(* CODESYS project EAS SCADA.library
   Author: EAS
   Placeholder: EAS SCADA
   Title: EAS SCADA
   Version: 1.0.4
   Company: ESCARRE AUTOMATIZACION Y SERVICIOS sl

Project tree, tasks and I/O mapping:
  libraries: Tc2_Standard, * (Beckhoff Automation GmbH); Tc2_System, * (Beckhoff Automation GmbH); Tc3_Module, * (Beckhoff Automation GmbH)
  DUTs/
    PE/
      data type E_Funcio
      data type PasCicle
      data type T_Compat
      data type T_funcio
      data type T_Sirena
  GVLs/
    global variables Batch
    global variables CONSTANTS
  POUs/
    BATCH/
      function block CarregarFuncionsActivesAlDB [ST]
      function block ComprobarFuncionsPas [ST]
      function block Inic_Func_Actv [ST]
      function block Parar_Func_FiFuncio [ST]
      function block Parar_Func_Incomp [ST]
      function block PararTotesLesFuncions [ST]
      function block Salt [ST]
      function block SaltDePasEnUnCicle [ST]
    GestioPE/
      function block Alarma_v01 [ST]
      function block FunBck_v01 [ST]
      function block Func_Activa_v01 [ST]
  VISUs/
*)

// DUTs/PE/E_Funcio
TYPE E_Funcio :
STRUCT

	Cd_Funcio:WORD;
	Actv_Funcio:BOOL;
	ParamFunc:ARRAY [1..Max_ParamFunc] OF WORD;

END_STRUCT
END_TYPE

// DUTs/PE/PasCicle
TYPE PasCicle :
STRUCT
	Pas:WORD;
	Funcio:E_Funcio;

END_STRUCT
END_TYPE

// DUTs/PE/T_Compat
TYPE T_Compat :
STRUCT

	Funcio1:WORD;  			(*Codi de la primera funcio*)
	Funcio2:WORD;  			(*Codi de la segona funcio*)

END_STRUCT
END_TYPE

// DUTs/PE/T_funcio
TYPE T_funcio :
STRUCT

	Cd_funcio:WORD;												(*Codi de la funció*)
	DesFuncio:STRING(16);										(*Descripció de la funció*)
	Background:BOOL;												(*Indicació per si la funció es en backgraund o no*)
	FinFunc:ARRAY [1..max_FinFunc] OF WORD;					(*Funcions que s'han d'acabar al començar aquesta*)

END_STRUCT
END_TYPE

// DUTs/PE/T_Sirena
TYPE T_Sirena :
STRUCT
	Actv:BOOL;
	Rearme:BOOL;
END_STRUCT
END_TYPE

// GVLs/Batch

VAR_GLOBAL RETAIN

(*=======================================	*)
(*					Estat del PE4							*)
(*=======================================	*)

(*Estat de PE4*)
	Func_Comp: ARRAY [1..Max_Compatibles] OF T_Compat;


(*=======================================	*)
(*			Variables de gestió de funcions				*)
(*=======================================	*)

(*Estat de lesFuncions *)
	Est_Func: ARRAY [1..Max_Funcions] OF E_Funcio;  		(*Estat actual de les funcions*)
	Est_F_PE4: ARRAY [1..Max_Funcions] OF E_Funcio;  		(*Estat de les funcions per les comunicacions del PE4*)
	Est_F_PE4_Ant: ARRAY [1..Max_Funcions] OF E_Funcio;  	(*Estat de les funcions per les comunicacions del PE4*)


(* *)
	Config_Func: ARRAY  [1..Max_Funcions] OF t_funcio;		(*Configuració de les funcios *)
	Config_Func_Ampl: ARRAY  [1..Max_Funcions] OF t_funcio_Ampl;		(*Configuració de les funcios ampliades*)
	Func_Actives: ARRAY [1..Max_Func_Pas] OF WORD;		(* DB que indica en automaatic les funcions que estan en marcha en automatic*)


(*=======================================	*)
(*			Variables de gestió de cicle					*)
(*=======================================	*)

(*Cicles*)
	Cicle0: ARRAY [1..max_PasCicle] OF PasCicle;  			(*Cicle Actual de treball*)
	CicleRebut: ARRAY [1..max_PasCicle] OF PasCicle;  		(*Cicle Rebut*)


(*=======================================	*)
(*					Alarmes								*)
(*=======================================	*)

	Alarmes:ARRAY[1..Max_Alarmes] OF T_Alarma;
	Sirena:ARRAY[1..Max_Alarmes] OF T_Sirena;


(*=======================================	*)
(*			Parametres fixes								*)
(*=======================================	*)

	ParamFixes:ARRAY[1..Max_ParamFixes] OF T_ParamFixe;


(*=======================================	*)
(*			Botons Auto/Man								*)
(*=======================================	*)

	PulsadorManual:BOOL;
	PulsadorAutomatic:BOOL;

(*=======================================	*)
(*			Marcas Internes								*)
(*=======================================	*)

	InicioCiclo:BOOL;


END_VAR


VAR_GLOBAL

(*=======================================	*)
(*			Maquina paralel 								*)
(*=======================================	*)

	TipoParalelo:WORD;
	MaquinaEnParalel:BOOL:=FALSE;
	Master:BOOL;
	Slave:BOOL;
	Pas_M:DWORD;
	Pas_S1:DWORD;
	Pas_S2:DWORD;
	Pas_S3:DWORD;
	Pas_S4:DWORD;
	Tipus_P:DWORD;
	Preparat_C_local:BOOL;
	He_C_local:BOOL;
	Ordre_C:BOOL;
	Ordre_C_Master:BOOL;
	Preparat_C_S1:BOOL;
	Preparat_C_S2:BOOL;
	Preparat_C_S3:BOOL;
	Preparat_C_S4:BOOL;
	He_C_S1:BOOL;
	He_C_S2:BOOL;
	He_C_S3:BOOL;
	He_C_S4:BOOL;
	Fi_C:BOOL;
	Fi_C_master:BOOL;



(*			CONSERVAR  COMPATIBILITAT				*)

	EsperaParalelPerSaltar:BOOL;
	SaltdePas:BOOL;


END_VAR

// GVLs/CONSTANTS

VAR_GLOBAL CONSTANT

(*=======================================	*)
(*			Carregar Constants						*)
(*=======================================	*)
	Max_Funcions:WORD:=64;
	Max_ParamFunc:WORD:=9;
	max_FinFunc:WORD:=5;
	max_PasCicle:WORD:=256;
	Max_Compatibles:WORD:=32;
	Max_Func_Pas:WORD:=12;
	Max_Alarmes:WORD:=128;
	Max_ParamFixes:WORD:=150;
	Max_DBFiFuncio: WORD:=320 ;				(* Es calcula com    (Max_Funcions*Max_FinFunc)   *)
	Max_ElementsCicle: WORD:=2816 ;		(* Es calcula com    (Max_PasCicle*(Max_ParamFunc+2))  *)
	Max_DBIncompatibles: WORD:=64;			(* Es calcula com    (Max_Compatibles*2)  *)
	Max_Inputs: WORD:=128;
	Max_Outputs: WORD:=128;
	Max_Analog: WORD:=32;
	Num_Prod_Dos:WORD:=10;         					(* Numero maximo de productos en una dosificación*)
	Max_Prod_Dos:WORD:=128;							(* Productos en una dosificadora*)
	Max_Valv_Dos:WORD:=128;							(* Valvulas en una dosificadora*)
END_VAR

// POUs/BATCH/CarregarFuncionsActivesAlDB
FUNCTION_BLOCK CarregarFuncionsActivesAlDB

(***********************************************************************
Aquest Bloc Carrega les Funcions actives al "DB d'estat de les funcions"
al "DB de funcions actives".   
************************************************************************)

VAR_INPUT
	EstatFuncions: ARRAY [1..max_funcions] OF E_Funcio;
END_VAR

VAR_OUTPUT
	FuncionsActives:ARRAY [1..Max_Func_Pas] OF WORD;
END_VAR

VAR
	Punter:WORD;
	PunterDB:WORD;
	inicialitzaDB: Inic_Func_Actv;
	DB_ple: BOOL;

END_VAR

inicialitzaDB(Func_Actv:= FuncionsActives);
DB_Ple:=FALSE;
punter:=1;
punterDB:=1;
WHILE (punter<=max_funcions)AND NOT(DB_Ple)
	DO
		IF EstatFuncions[punter].Actv_Funcio
			THEN
				FuncionsActives[PunterDB]:=EstatFuncions[punter].Cd_Funcio;
				PunterDB:=PunterDB+1;
				IF punterDB>Max_Func_Pas
					THEN
						DB_ple:=TRUE;
				END_IF
		END_IF
		punter:=punter+1;
END_WHILE

END_FUNCTION_BLOCK

// POUs/BATCH/Inic_Func_Actv
FUNCTION_BLOCK Inic_Func_Actv

(*********************************************************
Reinicia el DB de les funcions actives
***********************************************************)

VAR_IN_OUT
	Func_Actv: ARRAY [1..Max_Func_Pas] OF WORD;		(* DB que indica en automaatic les funcions que estan en marcha en automatic*)
END_VAR

VAR
	Punter: WORD;
END_VAR

Punter:=1;

REPEAT
	Func_Actv[punter]:=0;
	Punter:=Punter+1;
UNTIL
	Punter>Max_Func_Pas
END_REPEAT

END_FUNCTION_BLOCK

// POUs/BATCH/ComprobarFuncionsPas
FUNCTION_BLOCK ComprobarFuncionsPas

(************************************************************
Aquest Bloc Comproba les funcions actves que hi ha en aquest
pas i quan acaben dona l'ordr de canviar de pas.
**************************************************************)

VAR_INPUT
	Estat_F: ARRAY [1..Max_Funcions] OF E_Funcio;
	Tipus_F:ARRAY [1..Max_Funcions] OF T_Funcio;
	FuncionsActives:ARRAY [1..Max_Func_Pas] OF WORD;
END_VAR

VAR_OUTPUT
	AumentaPas:BOOL;
END_VAR

VAR
	Punter: WORD;
	Aumenta: BOOL;
	TempoPAS:TON;

END_VAR

(*Inicialitzar els punters*)
Punter:=1;
Aumenta:=TRUE;

REPEAT
	IF (FuncionsActives[Punter]<>0)AND((Estat_F[FuncionsActives[Punter]].Actv_Funcio=TRUE)AND(Tipus_F[FuncionsActives[Punter]].Background=FALSE))
		THEN
			Aumenta:=FALSE;
	END_IF
	Punter:=Punter+1;
UNTIL
	(Punter>Max_Func_Pas)OR(Aumenta=FALSE)
END_REPEAT

TempoPAS
	(IN:=Aumenta ,
	PT:=t#500ms ,
	Q=>AumentaPas ,
	ET=> );

END_FUNCTION_BLOCK

// POUs/BATCH/Parar_Func_FiFuncio
FUNCTION_BLOCK Parar_Func_FiFuncio

(**************************************************
Para les funcions del "DB de l'estat de funcions" 
depenen de la funcio de la entreda per "fifuncion"
***************************************************)

VAR_INPUT
	Tipus_Funcio:T_funcio;
END_VAR
VAR_OUTPUT
END_VAR
VAR_IN_OUT
	Estat_F: ARRAY [1..Max_Funcions] OF E_Funcio;
END_VAR
VAR
	PunterFiFunc:WORD;
	FuncioIncompat: WORD;
END_VAR

(*..................	Parar les funcions per fin función..................................	*)
PunterFiFunc:=1;
WHILE (PunterFiFunc <= max_FinFunc) DO
	FuncioIncompat :=Tipus_funcio.FinFunc[PunterFiFunc];
	IF FuncioIncompat <>0
		THEN
			Estat_F [FuncioIncompat].Actv_Funcio:=FALSE;
	END_IF
	PunterFiFunc:=PunterFiFunc+1;
END_WHILE

END_FUNCTION_BLOCK

// POUs/BATCH/Parar_Func_Incomp
FUNCTION_BLOCK Parar_Func_Incomp
(************************************************************
L'hi introduim una funció i el el bloc para les funcions del 
"DB estat de les funcions" depenen del 
"DB de compatibilitat"
**************************************************************)
VAR_INPUT
	Funcio:WORD;  (*Funcio que s'ha de parar*)
END_VAR

VAR_OUTPUT
END_VAR

VAR_IN_OUT
	DB_Comp:ARRAY [1..Max_Compatibles] OF T_Compat;
	Estat_F: ARRAY [1..Max_Funcions] OF E_Funcio;
END_VAR

VAR
	PunterEstat:WORD;
	PunterComp:WORD;
END_VAR

(*Mirar si hi ha alguna funció incompatible amb la nova funció*)
PunterEstat:=1;
PunterComp:=1;
REPEAT
	IF DB_Comp[PunterComp].Funcio1=Funcio
		THEN
			PunterEstat:=DB_Comp[PunterComp].Funcio2;
			Estat_F[PunterEstat].Actv_Funcio:=FALSE;
	END_IF
	PunterComp:=PunterComp+1;
UNTIL
	(PunterComp>Max_Compatibles)
END_REPEAT

END_FUNCTION_BLOCK

// POUs/BATCH/PararTotesLesFuncions
FUNCTION_BLOCK PararTotesLesFuncions
(********************************************************
Parar totes les funcions del "DB estat"
*********************************************************)
VAR_IN_OUT
	Estat_F: ARRAY [1..Max_Funcions] OF E_Funcio;
END_VAR

VAR
	Punter: WORD;
END_VAR

(*Inicialitzar els punters*)
Punter:=1;


WHILE (Punter <= Max_Funcions) DO
	IF Estat_F[Punter].Actv_Funcio=TRUE
		THEN
			Estat_F [Punter].Actv_Funcio:=FALSE;
	END_IF
	Punter:=Punter+1;
END_WHILE

END_FUNCTION_BLOCK

// POUs/BATCH/Salt
FUNCTION_BLOCK Salt
(************************************************************
Salta del "Pas inicial" al "Pas Final"  del  "BDCicle"
**************************************************************)
VAR_INPUT
	PasInicial:DWORD;
	PasFinal:DWORD;
END_VAR

VAR_IN_OUT


END_VAR

VAR

	FIFuncio:Parar_Func_FiFuncio;
	Incompatibles:Parar_Func_Incomp;
	PunterCicle:WORD;					(* Aquest valor marca la popsició del db de cicle on estem independent del pas de cicle *)
	T_Func_Act:T_Funcio;				(* Funcio que indica el punterCicle *)

	codi: WORD;

	Est_Func_0: ARRAY [1..Max_Funcions] OF E_Funcio;  		(*Estat de les funcions a cero per reiniciar l'estat*)
END_VAR

(*,,,,,,,,,,,,,,,,,,,,Carregar la posició inicial depenen si es salta desde:
				el pas cero: carerega d'un cicle nou
				un pas en concret: salt sobre el cicle que ja està carregat ,,,,,,,,,,,,,,,,,,,,,  *)

IF PasInicial=0
	THEN
		(*Posar Punter al primer pas*)
		PunterCicle:=1;
		(*Inicialitzar el estat de les funcions*)
		Est_Func:=Est_Func_0;
	ELSE
		(*Buscar Punter Cicle del pas inicial*)
		PunterCicle:=0;
		REPEAT
			PunterCicle := PunterCicle+1;
		UNTIL
			(((Cicle0[PunterCicle].Pas=PasInicial)AND(Cicle0[PunterCicle+1].Pas<>PasInicial)) OR (PunterCicle>=max_PasCicle))
		END_REPEAT
		PunterCicle := PunterCicle+1;      (*02/06/05*)
END_IF

(*,,,,,,,,,,,,,,,,,,,,Bucle de control,,,,,,,,,,,,,,,,,,,,,,,,,,,,,,,,,,,,,,,,,,,,,,,,,,,,,,,,,,,,,	*)

REPEAT
(*.................. Carregar la funció del pas............................................. *)
		codi:=Cicle0[PunterCicle].Funcio.Cd_Funcio;
		IF codi<>0 THEN
		T_Func_Act:=Config_Func[codi];
		END_IF
(*..................	Parar les funcions incompatibles..................................	*)
		Incompatibles(
			Funcio:=T_Func_Act.Cd_funcio ,
			DB_Comp:= Func_Comp ,
			Estat_F:= Est_Func );

(*..................	Activar si es en Background ........................................	*)
		IF T_Func_Act.Background=TRUE
			THEN
				Est_Func[T_Func_Act.Cd_Funcio] := Cicle0[PunterCicle].Funcio ; 	(*Carregar parametres*)
				Est_Func[T_Func_Act.Cd_Funcio].Actv_Funcio:=TRUE;			(*Posar la funció en actiu*)
		END_IF

(*..................	Parar les funcions per fin función..................................	*)
		FiFuncio(
			Tipus_Funcio:=  T_Func_Act ,
			 Estat_F:=Est_Func	 );

(*,,,,,,,,,,,,,,,,,,	Activar funció,,,,,,,,,,,,,,,,,,,,,,,,,,,,,,,,,,,,,,,,,,,,,,,,,,,,,,,,,,,,,,,,,,,	*)
		IF Cicle0[PunterCicle].Pas = PasFinal
			THEN
				Est_Func[T_Func_Act.Cd_Funcio] := Cicle0[PunterCicle].Funcio ;	(*Carregar parametres*)
				Est_Func[T_Func_Act.Cd_Funcio].Actv_Funcio := TRUE;			(*Posar la funció en actiu*)
		END_IF

(*,,,,,,,,,,,,,,,,,,Aumentar el Punter del cicle,,,,,,,,,,,,,,,,,,,,,,,,,,,,,,,,,,,,,,,,,,	*)
		PunterCicle := PunterCicle+1;

UNTIL
	(((Cicle0[PunterCicle].Pas <> PasFinal)AND(Cicle0[PunterCicle-1].Pas = PasFinal))
	OR(PunterCicle>max_PasCicle)
	OR(Cicle0[PunterCicle-1].Funcio.Cd_Funcio=0))
END_REPEAT

END_FUNCTION_BLOCK

// POUs/BATCH/SaltDePasEnUnCicle
FUNCTION_BLOCK SaltDePasEnUnCicle
(************************************************************
Salta del "Pas inicial" al "Pas Final"  del  "BDCicle"
**************************************************************)
VAR_INPUT
	PasInicial:DWORD;
	PasFinal:DWORD;
END_VAR

VAR_IN_OUT


END_VAR

VAR

	FIFuncio:Parar_Func_FiFuncio;
	Incompatibles:Parar_Func_Incomp;
	PunterCicle:WORD;					(* Aquest valor marca la popsició del db de cicle on estem independent del pas de cicle *)
	T_Func_Act:T_Funcio;				(* Funcio que indica el punterCicle *)

	codi: WORD;

	Est_Func_0: ARRAY [1..Max_Funcions] OF E_Funcio;  		(*Estat de les funcions a cero per reiniciar l'estat*)
END_VAR

(*,,,,,,,,,,,,,,,,,,,,Carregar la posició inicial depenen si es salta desde:
				el pas cero: carerega d'un cicle nou
				un pas en concret: salt sobre el cicle que ja està carregat ,,,,,,,,,,,,,,,,,,,,,  *)

IF PasInicial=0
	THEN
		(*Posar Punter al primer pas*)
		PunterCicle:=1;
		(*Inicialitzar el estat de les funcions*)
		Est_Func:=Est_Func_0;
	ELSE
		(*Buscar Punter Cicle del pas inicial*)
		PunterCicle:=0;
		REPEAT
			PunterCicle := PunterCicle+1;
		UNTIL
			(((Cicle0[PunterCicle].Pas=PasInicial)AND(Cicle0[PunterCicle+1].Pas<>PasInicial)) OR (PunterCicle>=max_PasCicle))
		END_REPEAT
		PunterCicle := PunterCicle+1;      (*02/06/05*)
END_IF

(*,,,,,,,,,,,,,,,,,,,,Bucle de control,,,,,,,,,,,,,,,,,,,,,,,,,,,,,,,,,,,,,,,,,,,,,,,,,,,,,,,,,,,,,	*)

REPEAT
(*.................. Carregar la funció del pas............................................. *)
		codi:=Cicle0[PunterCicle].Funcio.Cd_Funcio;
		IF codi<>0 THEN
		T_Func_Act:=Config_Func[codi];
		END_IF
(*..................	Parar les funcions incompatibles..................................	*)
		Incompatibles(
			Funcio:=T_Func_Act.Cd_funcio ,
			DB_Comp:= Func_Comp ,
			Estat_F:= Est_Func );

(*..................	Activar si es en Background ........................................	*)
		IF T_Func_Act.Background=TRUE
			THEN
				Est_Func[T_Func_Act.Cd_Funcio] := Cicle0[PunterCicle].Funcio ; 	(*Carregar parametres*)
				Est_Func[T_Func_Act.Cd_Funcio].Actv_Funcio:=TRUE;			(*Posar la funció en actiu*)
		END_IF

(*..................	Parar les funcions per fin función..................................
		FiFuncio(
			Tipus_Funcio:=  T_Func_Act ,
			 Estat_F:=Est_Func	 );										*)

(*,,,,,,,,,,,,,,,,,,	Activar funció,,,,,,,,,,,,,,,,,,,,,,,,,,,,,,,,,,,,,,,,,,,,,,,,,,,,,,,,,,,,,,,,,,,	*)
		IF Cicle0[PunterCicle].Pas = PasFinal
			THEN
				Est_Func[T_Func_Act.Cd_Funcio] := Cicle0[PunterCicle].Funcio ;	(*Carregar parametres*)
				Est_Func[T_Func_Act.Cd_Funcio].Actv_Funcio := TRUE;			(*Posar la funció en actiu*)
		END_IF

(*,,,,,,,,,,,,,,,,,,Aumentar el Punter del cicle,,,,,,,,,,,,,,,,,,,,,,,,,,,,,,,,,,,,,,,,,,	*)
		PunterCicle := PunterCicle+1;

UNTIL
	(((Cicle0[PunterCicle].Pas <> PasFinal)AND(Cicle0[PunterCicle-1].Pas = PasFinal))
	OR(PunterCicle>max_PasCicle)
	OR(Cicle0[PunterCicle-1].Funcio.Cd_Funcio=0))
END_REPEAT

END_FUNCTION_BLOCK

// POUs/GestioPE/Alarma_v01
FUNCTION_BLOCK Alarma_v01

(******************************************************
Aquest Bloc serveix per reactivar les senyals d'alarma
treballa amb el DB Sirena
********************************************************)

VAR_INPUT
END_VAR
VAR_OUTPUT
	ReactivaAlarma: BOOL;
	AlarmaActv: BOOL;
END_VAR

VAR_IN_OUT
END_VAR

VAR
	PolsA1:R_TRIG;
	PolsA2:R_TRIG;
	PolsA3:R_TRIG;
	PolsA4:R_TRIG;
	PolsA5:R_TRIG;
	PolsA6:R_TRIG;
	PolsA7:R_TRIG;
	PolsA8:R_TRIG;
	PolsA9:R_TRIG;
	PolsA10:R_TRIG;
	PolsA11:R_TRIG;
	PolsA12:R_TRIG;
	PolsA13:R_TRIG;
	PolsA14:R_TRIG;
	PolsA15:R_TRIG;
	PolsA16:R_TRIG;
	PolsA17:R_TRIG;
	PolsA18:R_TRIG;
	PolsA19:R_TRIG;
	PolsA20:R_TRIG;
	PolsA21:R_TRIG;
	PolsA22:R_TRIG;
	PolsA23:R_TRIG;
	PolsA24:R_TRIG;
	PolsA25:R_TRIG;
	PolsA26:R_TRIG;
	PolsA27:R_TRIG;
	PolsA28:R_TRIG;
	PolsA29:R_TRIG;
	PolsA30:R_TRIG;
	PolsA31:R_TRIG;
	PolsA32:R_TRIG;
	PolsA33:R_TRIG;
	PolsA34:R_TRIG;
	PolsA35:R_TRIG;
	PolsA36:R_TRIG;
	PolsA37:R_TRIG;
	PolsA38:R_TRIG;
	PolsA39:R_TRIG;
	PolsA40:R_TRIG;
	PolsA41:R_TRIG;
	PolsA42:R_TRIG;
	PolsA43:R_TRIG;
	PolsA44:R_TRIG;
	PolsA45:R_TRIG;
	PolsA46:R_TRIG;
	PolsA47:R_TRIG;
	PolsA48:R_TRIG;
	PolsA49:R_TRIG;
	PolsA50:R_TRIG;
	PolsA51:R_TRIG;
	PolsA52:R_TRIG;
	PolsA53:R_TRIG;
	PolsA54:R_TRIG;
	PolsA55:R_TRIG;
	PolsA56:R_TRIG;
	PolsA57:R_TRIG;
	PolsA58:R_TRIG;
	PolsA59:R_TRIG;
	PolsA60:R_TRIG;
	PolsA61:R_TRIG;
	PolsA62:R_TRIG;
	PolsA63:R_TRIG;
	PolsA64:R_TRIG;
	PolsA65:R_TRIG;
	PolsA66:R_TRIG;
	PolsA67:R_TRIG;
	PolsA68:R_TRIG;
	PolsA69:R_TRIG;
	PolsA70:R_TRIG;
	PolsA71:R_TRIG;
	PolsA72:R_TRIG;
	PolsA73:R_TRIG;
	PolsA74:R_TRIG;
	PolsA75:R_TRIG;
	PolsA76:R_TRIG;
	PolsA77:R_TRIG;
	PolsA78:R_TRIG;
	PolsA79:R_TRIG;
	PolsA80:R_TRIG;
	PolsA81:R_TRIG;
	PolsA82:R_TRIG;
	PolsA83:R_TRIG;
	PolsA84:R_TRIG;
	PolsA85:R_TRIG;
	PolsA86:R_TRIG;
	PolsA87:R_TRIG;
	PolsA88:R_TRIG;
	PolsA89:R_TRIG;
	PolsA90:R_TRIG;
	PolsA91:R_TRIG;
	PolsA92:R_TRIG;
	PolsA93:R_TRIG;
	PolsA94:R_TRIG;
	PolsA95:R_TRIG;
	PolsA96:R_TRIG;
	PolsA97:R_TRIG;
	PolsA98:R_TRIG;
	PolsA99:R_TRIG;
	PolsA100:R_TRIG;
	PolsA101:R_TRIG;
	PolsA102:R_TRIG;
	PolsA103:R_TRIG;
	PolsA104:R_TRIG;
	PolsA105:R_TRIG;
	PolsA106:R_TRIG;
	PolsA107:R_TRIG;
	PolsA108:R_TRIG;
	PolsA109:R_TRIG;
	PolsA110:R_TRIG;
	PolsA111:R_TRIG;
	PolsA112:R_TRIG;
	PolsA113:R_TRIG;
	PolsA114:R_TRIG;
	PolsA115:R_TRIG;
	PolsA116:R_TRIG;
	PolsA117:R_TRIG;
	PolsA118:R_TRIG;
	PolsA119:R_TRIG;
	PolsA120:R_TRIG;
	PolsA121:R_TRIG;
	PolsA122:R_TRIG;
	PolsA123:R_TRIG;
	PolsA124:R_TRIG;
	PolsA125:R_TRIG;
	PolsA126:R_TRIG;
	PolsA127:R_TRIG;
	PolsA128:R_TRIG;


	punter: WORD;
	punterA: WORD;
END_VAR

PolsA1(CLK:=Sirena[1].Actv , Q=>Sirena[1].Rearme);
PolsA2(CLK:=Sirena[2].Actv , Q=>Sirena[2].Rearme);
PolsA3(CLK:=Sirena[3].Actv , Q=>Sirena[3].Rearme);
PolsA4(CLK:=Sirena[4].Actv , Q=>Sirena[4].Rearme);
PolsA5(CLK:=Sirena[5].Actv , Q=>Sirena[5].Rearme);
PolsA6(CLK:=Sirena[6].Actv , Q=>Sirena[6].Rearme);
PolsA7(CLK:=Sirena[7].Actv , Q=>Sirena[7].Rearme);
PolsA8(CLK:=Sirena[8].Actv , Q=>Sirena[8].Rearme);
PolsA9(CLK:=Sirena[9].Actv , Q=>Sirena[9].Rearme);
PolsA10(CLK:=Sirena[10].Actv , Q=>Sirena[10].Rearme);
PolsA11(CLK:=Sirena[11].Actv , Q=>Sirena[11].Rearme);
PolsA12(CLK:=Sirena[12].Actv , Q=>Sirena[12].Rearme);
PolsA13(CLK:=Sirena[13].Actv , Q=>Sirena[13].Rearme);
PolsA14(CLK:=Sirena[14].Actv , Q=>Sirena[14].Rearme);
PolsA15(CLK:=Sirena[15].Actv , Q=>Sirena[15].Rearme);
PolsA16(CLK:=Sirena[16].Actv , Q=>Sirena[16].Rearme);
PolsA17(CLK:=Sirena[17].Actv , Q=>Sirena[17].Rearme);
PolsA18(CLK:=Sirena[18].Actv , Q=>Sirena[18].Rearme);
PolsA19(CLK:=Sirena[19].Actv , Q=>Sirena[19].Rearme);
PolsA20(CLK:=Sirena[20].Actv , Q=>Sirena[20].Rearme);
PolsA21(CLK:=Sirena[21].Actv , Q=>Sirena[21].Rearme);
PolsA22(CLK:=Sirena[22].Actv , Q=>Sirena[22].Rearme);
PolsA23(CLK:=Sirena[23].Actv , Q=>Sirena[23].Rearme);
PolsA24(CLK:=Sirena[24].Actv , Q=>Sirena[24].Rearme);
PolsA25(CLK:=Sirena[25].Actv , Q=>Sirena[25].Rearme);
PolsA26(CLK:=Sirena[26].Actv , Q=>Sirena[26].Rearme);
PolsA27(CLK:=Sirena[27].Actv , Q=>Sirena[27].Rearme);
PolsA28(CLK:=Sirena[28].Actv , Q=>Sirena[28].Rearme);
PolsA29(CLK:=Sirena[29].Actv , Q=>Sirena[29].Rearme);
PolsA30(CLK:=Sirena[30].Actv , Q=>Sirena[30].Rearme);
PolsA31(CLK:=Sirena[31].Actv , Q=>Sirena[31].Rearme);
PolsA32(CLK:=Sirena[32].Actv , Q=>Sirena[32].Rearme);
PolsA33(CLK:=Sirena[33].Actv , Q=>Sirena[33].Rearme);
PolsA34(CLK:=Sirena[34].Actv , Q=>Sirena[34].Rearme);
PolsA35(CLK:=Sirena[35].Actv , Q=>Sirena[35].Rearme);
PolsA36(CLK:=Sirena[36].Actv , Q=>Sirena[36].Rearme);
PolsA37(CLK:=Sirena[37].Actv , Q=>Sirena[37].Rearme);
PolsA38(CLK:=Sirena[38].Actv , Q=>Sirena[38].Rearme);
PolsA39(CLK:=Sirena[39].Actv , Q=>Sirena[39].Rearme);
PolsA40(CLK:=Sirena[40].Actv , Q=>Sirena[40].Rearme);
PolsA41(CLK:=Sirena[41].Actv , Q=>Sirena[41].Rearme);
PolsA42(CLK:=Sirena[42].Actv , Q=>Sirena[42].Rearme);
PolsA43(CLK:=Sirena[43].Actv , Q=>Sirena[43].Rearme);
PolsA44(CLK:=Sirena[44].Actv , Q=>Sirena[44].Rearme);
PolsA45(CLK:=Sirena[45].Actv , Q=>Sirena[45].Rearme);
PolsA46(CLK:=Sirena[46].Actv , Q=>Sirena[46].Rearme);
PolsA47(CLK:=Sirena[47].Actv , Q=>Sirena[47].Rearme);
PolsA48(CLK:=Sirena[48].Actv , Q=>Sirena[48].Rearme);
PolsA49(CLK:=Sirena[49].Actv , Q=>Sirena[49].Rearme);
PolsA50(CLK:=Sirena[50].Actv , Q=>Sirena[50].Rearme);
PolsA51(CLK:=Sirena[51].Actv , Q=>Sirena[51].Rearme);
PolsA52(CLK:=Sirena[52].Actv , Q=>Sirena[52].Rearme);
PolsA53(CLK:=Sirena[53].Actv , Q=>Sirena[53].Rearme);
PolsA54(CLK:=Sirena[54].Actv , Q=>Sirena[54].Rearme);
PolsA55(CLK:=Sirena[55].Actv , Q=>Sirena[55].Rearme);
PolsA56(CLK:=Sirena[56].Actv , Q=>Sirena[56].Rearme);
PolsA57(CLK:=Sirena[57].Actv , Q=>Sirena[57].Rearme);
PolsA58(CLK:=Sirena[58].Actv , Q=>Sirena[58].Rearme);
PolsA59(CLK:=Sirena[59].Actv , Q=>Sirena[59].Rearme);
PolsA60(CLK:=Sirena[60].Actv , Q=>Sirena[60].Rearme);
PolsA61(CLK:=Sirena[61].Actv , Q=>Sirena[61].Rearme);
PolsA62(CLK:=Sirena[62].Actv , Q=>Sirena[62].Rearme);
PolsA63(CLK:=Sirena[63].Actv , Q=>Sirena[63].Rearme);
PolsA64(CLK:=Sirena[64].Actv , Q=>Sirena[64].Rearme);
PolsA65(CLK:=Sirena[65].Actv , Q=>Sirena[65].Rearme);
PolsA66(CLK:=Sirena[66].Actv , Q=>Sirena[66].Rearme);
PolsA67(CLK:=Sirena[67].Actv , Q=>Sirena[67].Rearme);
PolsA68(CLK:=Sirena[68].Actv , Q=>Sirena[68].Rearme);
PolsA69(CLK:=Sirena[69].Actv , Q=>Sirena[69].Rearme);
PolsA70(CLK:=Sirena[70].Actv , Q=>Sirena[70].Rearme);
PolsA71(CLK:=Sirena[71].Actv , Q=>Sirena[71].Rearme);
PolsA72(CLK:=Sirena[72].Actv , Q=>Sirena[72].Rearme);
PolsA73(CLK:=Sirena[73].Actv , Q=>Sirena[73].Rearme);
PolsA74(CLK:=Sirena[74].Actv , Q=>Sirena[74].Rearme);
PolsA75(CLK:=Sirena[75].Actv , Q=>Sirena[75].Rearme);
PolsA76(CLK:=Sirena[76].Actv , Q=>Sirena[76].Rearme);
PolsA77(CLK:=Sirena[77].Actv , Q=>Sirena[77].Rearme);
PolsA78(CLK:=Sirena[78].Actv , Q=>Sirena[78].Rearme);
PolsA79(CLK:=Sirena[79].Actv , Q=>Sirena[79].Rearme);
PolsA80(CLK:=Sirena[80].Actv , Q=>Sirena[80].Rearme);
PolsA81(CLK:=Sirena[81].Actv , Q=>Sirena[81].Rearme);
PolsA82(CLK:=Sirena[82].Actv , Q=>Sirena[82].Rearme);
PolsA83(CLK:=Sirena[83].Actv , Q=>Sirena[83].Rearme);
PolsA84(CLK:=Sirena[84].Actv , Q=>Sirena[84].Rearme);
PolsA85(CLK:=Sirena[85].Actv , Q=>Sirena[85].Rearme);
PolsA86(CLK:=Sirena[86].Actv , Q=>Sirena[86].Rearme);
PolsA87(CLK:=Sirena[87].Actv , Q=>Sirena[87].Rearme);
PolsA88(CLK:=Sirena[88].Actv , Q=>Sirena[88].Rearme);
PolsA89(CLK:=Sirena[89].Actv , Q=>Sirena[89].Rearme);
PolsA90(CLK:=Sirena[90].Actv , Q=>Sirena[90].Rearme);
PolsA91(CLK:=Sirena[91].Actv , Q=>Sirena[91].Rearme);
PolsA92(CLK:=Sirena[92].Actv , Q=>Sirena[92].Rearme);
PolsA93(CLK:=Sirena[93].Actv , Q=>Sirena[93].Rearme);
PolsA94(CLK:=Sirena[94].Actv , Q=>Sirena[94].Rearme);
PolsA95(CLK:=Sirena[95].Actv , Q=>Sirena[95].Rearme);
PolsA96(CLK:=Sirena[96].Actv , Q=>Sirena[96].Rearme);
PolsA97(CLK:=Sirena[97].Actv , Q=>Sirena[97].Rearme);
PolsA98(CLK:=Sirena[98].Actv , Q=>Sirena[98].Rearme);
PolsA99(CLK:=Sirena[99].Actv , Q=>Sirena[99].Rearme);
PolsA100(CLK:=Sirena[100].Actv , Q=>Sirena[100].Rearme);
PolsA101(CLK:=Sirena[101].Actv , Q=>Sirena[101].Rearme);
PolsA102(CLK:=Sirena[102].Actv , Q=>Sirena[102].Rearme);
PolsA103(CLK:=Sirena[103].Actv , Q=>Sirena[103].Rearme);
PolsA104(CLK:=Sirena[104].Actv , Q=>Sirena[104].Rearme);
PolsA105(CLK:=Sirena[105].Actv , Q=>Sirena[105].Rearme);
PolsA106(CLK:=Sirena[106].Actv , Q=>Sirena[106].Rearme);
PolsA107(CLK:=Sirena[107].Actv , Q=>Sirena[107].Rearme);
PolsA108(CLK:=Sirena[108].Actv , Q=>Sirena[108].Rearme);
PolsA109(CLK:=Sirena[109].Actv , Q=>Sirena[109].Rearme);
PolsA110(CLK:=Sirena[110].Actv , Q=>Sirena[110].Rearme);
PolsA111(CLK:=Sirena[111].Actv , Q=>Sirena[111].Rearme);
PolsA112(CLK:=Sirena[112].Actv , Q=>Sirena[112].Rearme);
PolsA113(CLK:=Sirena[113].Actv , Q=>Sirena[113].Rearme);
PolsA114(CLK:=Sirena[114].Actv , Q=>Sirena[114].Rearme);
PolsA115(CLK:=Sirena[115].Actv , Q=>Sirena[115].Rearme);
PolsA116(CLK:=Sirena[116].Actv , Q=>Sirena[116].Rearme);
PolsA117(CLK:=Sirena[117].Actv , Q=>Sirena[117].Rearme);
PolsA118(CLK:=Sirena[118].Actv , Q=>Sirena[118].Rearme);
PolsA119(CLK:=Sirena[119].Actv , Q=>Sirena[119].Rearme);
PolsA120(CLK:=Sirena[120].Actv , Q=>Sirena[120].Rearme);
PolsA121(CLK:=Sirena[121].Actv , Q=>Sirena[121].Rearme);
PolsA122(CLK:=Sirena[122].Actv , Q=>Sirena[122].Rearme);
PolsA123(CLK:=Sirena[123].Actv , Q=>Sirena[123].Rearme);
PolsA124(CLK:=Sirena[124].Actv , Q=>Sirena[124].Rearme);
PolsA125(CLK:=Sirena[125].Actv , Q=>Sirena[125].Rearme);
PolsA126(CLK:=Sirena[126].Actv , Q=>Sirena[126].Rearme);
PolsA127(CLK:=Sirena[127].Actv , Q=>Sirena[127].Rearme);
PolsA128(CLK:=Sirena[128].Actv , Q=>Sirena[128].Rearme);


ReactivaAlarma:=FALSE;
punter:=1;
WHILE (punter<=Max_Alarmes)AND NOT(ReactivaAlarma) DO
	IF Sirena[punter].Rearme THEN
		ReactivaAlarma:=TRUE;
	END_IF
	punter:=punter+1;
END_WHILE


AlarmaActv:=FALSE;
punterA:=1;
WHILE (punterA<=Max_Alarmes)AND NOT(AlarmaActv) DO
	IF Sirena[punterA].Actv THEN
		AlarmaActv:=TRUE;
	END_IF
	punterA:=punterA+1;
END_WHILE

END_FUNCTION_BLOCK

// POUs/GestioPE/FunBck_v01
FUNCTION_BLOCK FunBck_v01
VAR_INPUT
END_VAR

VAR_OUTPUT
	funcioBck: BOOL;
END_VAR


VAR
	punter: WORD;
END_VAR

punter:=1;
funcioBck:=FALSE;

WHILE ((punter<= Max_Funcions)AND NOT(FuncioBck)) DO
	IF ((Est_func[punter].Actv_funcio)AND NOT(Config_Func[punter].Background))
		THEN
			FuncioBck:=TRUE;
	END_IF
	punter:=punter+1;
END_WHILE

END_FUNCTION_BLOCK

// POUs/GestioPE/Func_Activa_v01
FUNCTION_BLOCK Func_Activa_v01
VAR_INPUT
	EstatFunc:ARRAY [1..Max_Funcions] OF E_Funcio;
END_VAR
VAR_OUTPUT
	FuncionsActives:BOOL;
END_VAR
VAR
	a: WORD;
END_VAR

(*Inicialitza el punter*)
a:=1;
FuncionsActives:=FALSE;
REPEAT
	IF EstatFunc[a].Actv_Funcio=TRUE
		THEN
			FuncionsActives:=TRUE;
	END_IF
	a:=a+1;
UNTIL
(a>Max_Funcions)OR(FuncionsActives=TRUE)
END_REPEAT

END_FUNCTION_BLOCK
